PROGRAM NeutronFactoryStates
VAR
//Define all necessary variables for your application
	eNeutronFactoryState: E_NeutronFactoryStates := E_NeutronFactoryStates.Disabled;
END_VAR

CASE eNeutronFactoryState OF
	
	E_NeutronFactoryStates.Disabled:
		GVL.astAxes[MAIN.hmiAxisSelection].stControl.bEnable := FALSE;
	
	
	E_NeutronFactoryStates.Maintenance:
		GVL.astAxes[MAIN.hmiAxisSelection].stControl.bEnable := FALSE;
	
	
	E_NeutronFactoryStates.StartUp:
		GVL.astAxes[MAIN.hmiAxisSelection].stControl.bEnable := FALSE;
	
	
	E_NeutronFactoryStates.CoolingDown:
		GVL.astAxes[MAIN.hmiAxisSelection].stControl.bEnable := FALSE;
	
	
	E_NeutronFactoryStates.NotConfirmedReady:
		GVL.astAxes[MAIN.hmiAxisSelection].stControl.bEnable := FALSE;
	
	
	E_NeutronFactoryStates.ConfirmedReady:
		GVL.astAxes[MAIN.hmiAxisSelection].stControl.bEnable := TRUE;
		
END_CASE

END_PROGRAM

(* stored: Version 1.1.0.1, ProductVersion 3.1.4024.10
   POU NeutronFactoryStates: Id {d43beee5-2cf4-48df-b5fd-a87d1d36e622}, SpecialFunc None *)
